Universal Robots URScript: Project1pick4.script

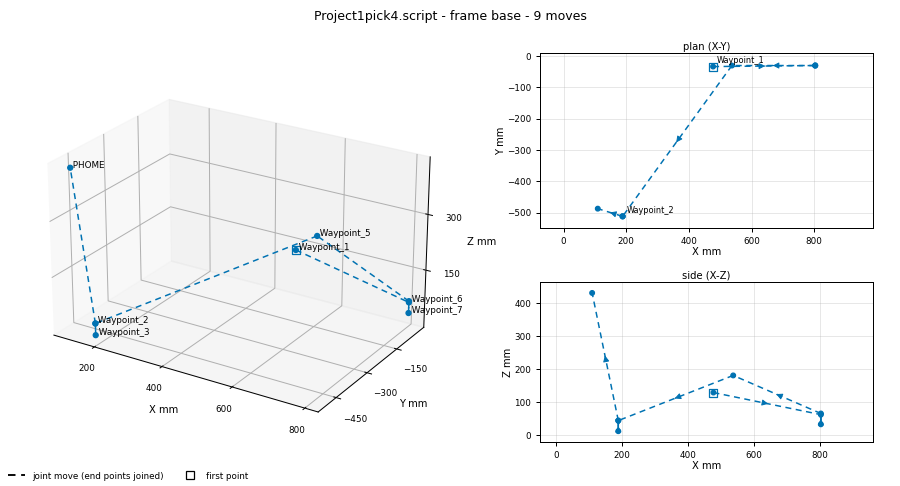
[picture p0: tool path of Project1pick4.script in frame base, 9 of 9 moves have a stored position in this frame; points joined in program order, loops and branches not executed]
def Project1pick4():
  set_tool_voltage(0)
  modbus_add_signal("127.0.0.1", 255, 1, 2, "MODBUS_1", False)
  modbus_set_signal_update_frequency("MODBUS_1", 10)
  modbus_add_signal("127.0.0.1", 255, 128, 0, "atLocation", False)
  modbus_set_signal_update_frequency("atLocation", 10)
  modbus_add_signal("10.241.34.56", 1, 1009, 3, "MODBUS_2", False)
  modbus_set_signal_update_frequency("MODBUS_2", 10)
  modbus_set_runstate_dependent_choice("MODBUS_2",0)
  set_safety_mode_transition_hardness(0)
  set_gravity([0.0, 0.0, 9.82])
  set_tcp(p[0.0,0.0,0.0,0.0,0.0,0.0])
  set_payload(1.0)
  step_count_9dcd0ba1_d11b_42b8_b275_8d807a8411d8 = 0.0
  thread Step_Counter_Thread_544c9fd5_7f06_4e61_a5b9_45d0981bf979():
    while (True):
      step_count_9dcd0ba1_d11b_42b8_b275_8d807a8411d8 = step_count_9dcd0ba1_d11b_42b8_b275_8d807a8411d8 + 1.0
      sync()
    end
  end
  run Step_Counter_Thread_544c9fd5_7f06_4e61_a5b9_45d0981bf979()
  set_standard_analog_input_domain(0, 1)
  set_standard_analog_input_domain(1, 1)
  set_tool_analog_input_domain(0, 0)
  set_tool_analog_input_domain(1, 0)
  set_analog_outputdomain(0, 0)
  set_analog_outputdomain(1, 0)
  set_input_actions_to_default()
  $ 1 "Robot Program"
  $ 2 "MoveJ"
  $ 3 "Waypoint_1" "breakAfter"
  movej(get_inverse_kin(p[.477217597624, -.033357379175, .129571503542, 2.226070920873, -2.211954177679, .005486199633], qnear=[2.842435121536255, -1.3189814726458948, 2.147374153137207, -2.4006994406329554, -1.5754440466510218, -0.3055227438556116]), a=1.3962634015954636, v=1.0471975511965976)
  $ 4 "Waypoint_6" "breakAfter"
  movej(get_inverse_kin(p[.803263884866, -.030050835915, .062587148046, 2.226059809870, -2.212020033750, .005679732930], qnear=[2.9684903621673584, -0.5888894240008753, 1.0668764114379883, -2.0498207251178187, -1.5756357351886194, -0.17943174043764287]), a=1.3962634015954636, v=1.0471975511965976)
  $ 5 "Waypoint_7" "breakAfter"
  movej(get_inverse_kin(p[.803243910290, -.030061005087, .033167975852, 2.225970237544, -2.211849555829, .005397257668], qnear=[2.9684784412384033, -0.5510314146624964, 1.0750923156738281, -2.0956419149981897, -1.575683895741598, -0.1794799009906214]), a=1.3962634015954636, v=1.0471975511965976)
  $ 6 "Wait: 0.5"
  sleep(0.5)
  $ 7 "Set DO[0]=On"
  set_standard_digital_out(0, True)
  $ 8 "Wait: 0.5"
  sleep(0.5)
  $ 9 "Waypoint_4" "breakAfter"
  movej(get_inverse_kin(p[.803271764079, -.030057233278, .066011026230, 2.226005484527, -2.211886220489, .005544952177], qnear=[2.9684903621673584, -0.5930669943438929, 1.065424919128418, -2.0440452734576624, -1.575695816670553, -0.1794675032245081]), a=1.3962634015954636, v=1.0471975511965976)
  $ 10 "Waypoint_5" "breakAfter"
  movej(get_inverse_kin(p[.537258936932, -.030094581372, .181531098877, 2.225919936588, -2.211812794864, .005424506883], qnear=[2.8821353912353516, -1.2909801642047327, 1.9299049377441406, -2.2109087149249476, -1.5756600538836878, -0.265817944203512]), a=1.3962634015954636, v=1.0471975511965976)
  $ 11 "Waypoint_2" "breakAfter"
  movej(get_inverse_kin(p[.188485305729, -.511480707990, .044451097170, 2.226120019575, -2.211714387572, .005633065904], qnear=[1.7223751544952393, -1.0243294874774378, 2.005359172821045, -2.5568226019488733, -1.5715130011187952, -1.425711456929342]), a=1.3962634015954636, v=1.0471975511965976)
  $ 12 "Waypoint_3" "breakAfter"
  movej(get_inverse_kin(p[.188430556532, -.511438580630, .012275395263, 2.226022424907, -2.211803209098, .005552531914], qnear=[1.7222912311553955, -0.9532488028155726, 2.0100016593933105, -2.6325085798846644, -1.5715487639056605, -1.425711456929342]), a=1.3962634015954636, v=1.0471975511965976)
  $ 13 "Wait: 0.5"
  sleep(0.5)
  $ 14 "Set DO[0]=Off"
  set_standard_digital_out(0, False)
  $ 15 "Wait: 0.5"
  sleep(0.5)
  $ 16 "Waypoint_2" "breakAfter"
  movej(get_inverse_kin(p[.188485305729, -.511480707990, .044451097170, 2.226120019575, -2.211714387572, .005633065904], qnear=[1.7223751544952393, -1.0243294874774378, 2.005359172821045, -2.5568226019488733, -1.5715130011187952, -1.425711456929342]), a=1.3962634015954636, v=1.0471975511965976)
  $ 17 "PHOME" "breakAfter"
  movej(get_inverse_kin(p[.109126925635, -.486916656758, .431880490887, .000103389846, 3.141554489202, -.000205683921], qnear=[1.5707424879074097, -1.570796314870016, 1.5707731246948242, -1.5709040800677698, -1.5707581678973597, 1.1984225238848012E-5]), a=1.3962634015954636, v=1.0471975511965976)
end
